// TIA Portal V17 export
// export: Created 2024-09-03T21:54:50.1013354Z, ExportSetting WithDefaults, DisplayName Totally Integrated Automation Portal, DisplayVersion V17 Update 7, DisplayName TIA Portal Openness, DisplayVersion V17 Update 7, DisplayName TIA Portal Version Control Interface, DisplayVersion V17, DisplayName SINAMICS Startdrive Advanced, DisplayVersion V17 SP2, DisplayName SINAMICS Startdrive G110M, G120, G120C, G120D, G120P, G115D, DisplayVersion V17 SP2, DisplayName SINAMICS Startdrive G130, G150, S120, S150, SINAMICS MV, S210, DisplayVersion V17 SP2, DisplayName STEP 7 Professional, DisplayVersion V17 Update 7, DisplayName STEP 7 Safety, DisplayVersion V17 Update 6, DisplayName WinCC Advanced / Unified PC, DisplayVersion V17 Update 7
DATA_BLOCK "DiagnosticConfigured"   // DB38
{ S7_Optimized_Access := 'TRUE' }
VERSION : 0.1
// stored: AutoNumber true, DBAccessibleFromOPCUA true, DBAccessibleFromWebserver true, IsOnlyStoredInLoadMemory false, IsRetainMemResEnabled false, IsWriteProtectedInAS false, MemoryReserve 100
   VAR
      Adresses : Array[1..255] of Int;
      Errors : Array[1..255] of Bool;
      Exists : Array[1..255] of Bool;
      States : Array[1..255] of Int;
      Updated : Bool := FALSE;
   END_VAR
BEGIN
   Adresses[1] := 11;
   Adresses[2] := 31;
   Adresses[3] := 32;
   Adresses[4] := 33;
   Adresses[5] := 34;
   Adresses[6] := 41;
   Adresses[7] := 61;
   Adresses[8] := 62;
   Adresses[9] := 63;
   Adresses[10] := 64;
   Adresses[11] := 65;
   Adresses[12] := 66;
   Adresses[13] := 68;
   Adresses[14] := 69;
   Adresses[15] := 70;
   Adresses[16] := 71;
   Adresses[17] := 73;
   Adresses[18] := 74;
   Adresses[19] := 91;
   Adresses[20..255] := 0;
   Errors[1..255] := FALSE;
   Exists[1..19] := TRUE;
   Exists[20..255] := FALSE;
   States[1..19] := 1;
   States[20..255] := 0;
END_DATA_BLOCK
